Yaskawa INFORM job: AAA.JBI

/JOB
//NAME AAA
//POS
///NPOS 2,0,0,0,0,0
C00000=6125,45284,-11571,23593,-45778,-28966
C00001=6338,38591,-18707,24005,-44956,-29286
//INST
///DATE 2023/02/07 14:07
///ATTR SC,RW
///GROUP1 RB1
NOP
MOVL C00000 V=10.0 PL=8
MOVL C00001 V=10.0 PL=0
END
